(* Schneider Machine Expert - Basic project PLO, file version 1.8.0.0 *)
(* ProjectInformations: Name=New project *)

HARDWARE
  Cpu 0: TM221CE16R
  EthernetConfiguration: NetworkName=M221, IpAllocationMode=FixedAddress, IpAddress=0.0.0.0, SubnetMask=0.0.0.0
  SerialLineConfiguration: Baud=Baud19200, Parity=ParityEven, DataBits=DataBits8, StopBits=StopBits1, PhysicalMedium=PhysicalMediumRs485, TransmissionMode=TransmissionModeModbusRtu, SlaveId=1, Addressing=SlaveAddressing
  MastTask: UsePeriodScanMode=false, PeriodScan=100
  FastTask: Period=255
  CpuBehavior: StartingMode=StartAsPreviousState, AutoSaveRamOnEeprom=true, WatchdogPeriod=250

SYMBOLS  (address, symbol, comment, settings)

POU New POU
  (* SectionNumber=1 *)

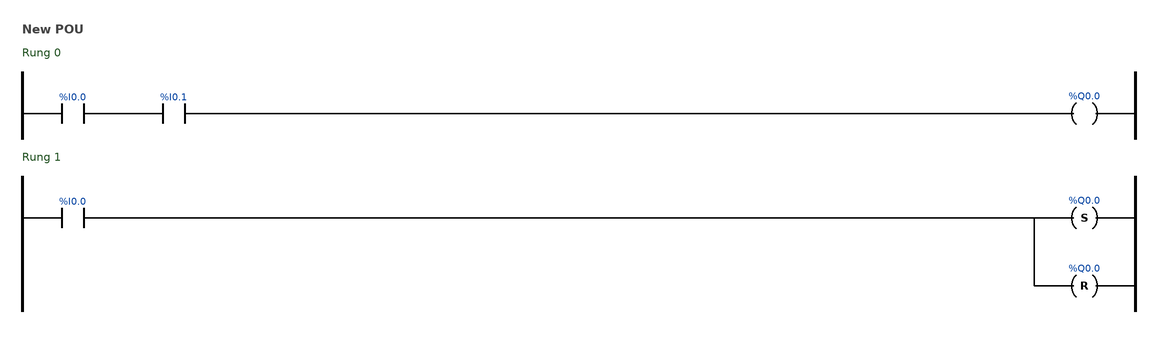

// Rung 0
  LD %I0.0
  AND %I0.1
  ST %Q0.0
  // as ST:
  //   %Q0.0 := %I0.0 AND %I0.1;

// Rung 1
  LD %I0.0
  S %Q0.0
  R %Q0.0
  // as ST:
  //   IF %I0.0 THEN %Q0.0 := TRUE; END_IF;
  //   IF %I0.0 THEN %Q0.0 := FALSE; END_IF;
